Staubli VAL3: sendData.pgx

public program sendData()
  local num l_nRetVal
begin
  userPage()
  while (true)
    nTrsfOut[0]=trShiftOut.x
    nTrsfOut[1]=trShiftOut.y
    nTrsfOut[2]=trShiftOut.z
    nTrsfOut[3]=trShiftOut.rx
    nTrsfOut[4]=trShiftOut.ry
    nTrsfOut[5]=trShiftOut.rz

    toBinary(nTrsfOut,6,"-4l",nByteOut)
    l_nRetVal = sioSet(siTcpSender,nByteOut)
    if (l_nRetVal == -1)
      putln("Not connected")
    endIf
  endWhile
end
